TEXTLIST TextList1
  0 = 'Auto Mode'
  1 = 'Manual Mode'
   = ''
END_TEXTLIST

(* stored: Version 1.1.0.1, ProductVersion 3.1.4024.15
   TextList TextList1: Id {c05cb724-522e-432e-90ae-4d66f24a59f2} *)
